FUNCTION UpdateTimeStampWithSystemTime : BOOL
VAR_INPUT
	stEvent : REFERENCE TO ST_Event;
END_VAR
VAR
	fbGetSystemTime  : GETSYSTEMTIME;
	stFileTime : T_FILETIME;
END_VAR

fbGetSystemTime(timeLoDW => stFiletime.dwLowDateTime,
				 timeHiDW => stFileTime.dwHighDateTime);
stEvent.dtTimeStamp := FILETIME_TO_DT(fileTime := stFileTime);

END_FUNCTION

(* stored: Version 1.1.0.1, ProductVersion 3.1.4024.16
   POU UpdateTimeStampWithSystemTime: Id {be573526-e4b8-4b40-bc83-dbbbda21196c}, SpecialFunc None *)
